{attribute 'qualified_only'}
{attribute 'strict'}
TYPE E_CX_NetworkInfoState : (
	IDLE,
	GETDEVICETYPE,
	GETHOSTNAME,
	GETLOCALAMSNETID,
	GETADAPTERINFO,
	GETDNSINFO,
	GETSNTPSERVER,
	GETSNTPTIME,
	DONE
);
END_TYPE

(* stored: Version 1.1.0.1
   DUT E_CX_NetworkInfoState: Id {048fec68-b7fb-4bba-8888-127a10c275d4} *)
